Omron CX-Programmer project NewProject (CX-Programmer 9.66)

# PLC LQK19011ICM: CP1H XA
I/O table (CPU CP1H-XA40DR-A): rack 0 slot 0 CJ1W-SCU21

## Global symbols (name address type ; comment)
0.04 BOOL  ; SPARE
0.05 BOOL  ; SPARE
0.07 BOOL  ; VERTICAL.AXIS.DOWN.LIMT
0.08 BOOL  ; C0A
0.09 BOOL  ; C0B
0.11 BOOL  ; SAW.SOFT.START.FAULT
10 CHANNEL  ; Initialize the High Speed Encoder Channel to 0
100.00 BOOL  ; WATER.VALVE
100.01 BOOL  ; SOFT.START.RUN
100.02 BOOL  ; VERTICAL.AXIS.RAISE
100.03 BOOL  ; VERTICAL.AXIS.LOWER
100.04 BOOL  ; TRANSVERSE.AXIS.FORWARD
100.05 BOOL  ; TRANSVERSE.AXIS.REVERSE
100.06 BOOL  ; VERTICAL.AXIS.SPEED.SELECT
101.00 BOOL  ; SOFT.START.STOP
101.01 BOOL  ; ALARM
101.02 BOOL  ; LONG.AXIS.MASTER.DRV.INDEX.COMMAND
101.03 BOOL  ; VERTICAL.AXIS.BRAKE
101.04 BOOL  ; LONG.AXIS.MASTER.DRV.JOG.LEFT
101.05 BOOL  ; LONG.AXIS.MASTER.DRV.JOG.RIGHT
101.06 BOOL  ; LONG.AXIS.MASTER.DRV.INITIATE.HOME.MOVE
101.07 BOOL  ; LASER.ON
1.00 BOOL  ; WATER.FLOW.SWITCH
1.02 BOOL  ; SPARE
1.03 BOOL  ; PHOTOCELL_GAUCHE
1.04 BOOL  ; PHOTOCELL_DROIT
1.05 BOOL  ; TRANSVERSE.AXIS.HOME.PROXIMITY
1.06 BOOL  ; TRANSVERSE.AXIS.FORWARD.LIMT.PROXIMITY
1.07 BOOL  ; VERTICAL.AXIS.HOME.PROXIMITY
1.08 BOOL  ; VERTICAL.AXIS.FORWARD.LIMIT
1.12 BOOL  ; INCONNU
1.15 BOOL  ; DELETE
200 CHANNEL  ; ANALOG.INPUT1.SAW.CURRENT
210 CHANNEL  ; TRANSVERSE.AXIS.VELOCITY.REFERENCE
294 CHANNEL  ; RG3_FST_CUT
302 CHANNEL  ; Axis Long first Status Word
302.08 BOOL  ; LONG.AXIS.MASTER.STATUS.DRV.NEGLIM
302.09 BOOL  ; LONG.AXIS.MASTER.STATUS.DRV.POSLIM
302.13 BOOL  ; LONG.AXIS.MASTER.STATUS.DRV.JOGANYCMDCOMP
302.14 BOOL  ; LONG.AXIS.MASTER.STATUS.ABSPOSVAL
303 CHANNEL  ; Axis Long second status Word
303.00 BOOL  ; LONG.AXIS.MASTER.STATUS.DRV.INDEX0.LIMDISTHIT
303.01 BOOL  ; LONG.AXIS.MASTER.STATUS.DRV.INDEX0.CMD.INPRGRS
303.02 BOOL  ; LONG.AXIS.MASTER.STATUS.DRV.INDEX0.CMD.COMPLETE
303.03 BOOL  ; LONG.AXIS.MASTER.STATUS.DRV.INDEX0.PLSSTATUS
303.04 BOOL  ; LONG.AXIS.MASTER.STATUS.DRV.INDEX0.ACCELLERATING
303.05 BOOL  ; LONG.AXIS.MASTER.STATUS.DRV.INDEX0.ATVEL
303.06 BOOL  ; LONG.AXIS.MASTER.STATUS.DRV.INDEX0.DECELLERATING
303.07 BOOL  ; LONG.AXIS.MASTER.STATUS.DRV.INDEX.ANYCOMDCOMPLETE
303.08 BOOL  ; LONG.AXIS.MASTER.STATUS.DRV.PGMANYACTIVE
303.09 BOOL  ; LONG.AXIS.MASTER.STATUS.DRV.PGMANYCOMPLETE
303.10 BOOL  ; LONG.AXIS.MASTER.STATUS.DRV.PGM0.PGMRUNNING
303.11 BOOL  ; LONG.AXIS.MASTER.STATUS.DRV.PGM0.PGMCOMPLETE
304 CHANNEL  ; Axis Long third Status Word
304.00 BOOL  ; LONG.AXIS.MASTER.STATUS.DRV.ERROR.ERRORED
304.01 BOOL  ; LONG.AXIS.MASTER.STATUS.DRV.ERROR.SPDRIVETRIPACTIVE
304.02 BOOL  ; LONG.AXIS.MASTER.STATUS.DRV.ERROR.EZMOTION.WATCHDOG
304.03 BOOL  ; LONG.AXIS.MASTER.STATUS.DRV.ERROR.EZMOTION.INVALIDCONFIG
304.04 BOOL  ; LONG.AXIS.MASTER.STATUS.DRV.ERROR.EZMOTION.NVMINVALD
304.05 BOOL  ; LONG.AXIS.MASTER.STATUS.DRV.ERROR.EZMOTION.PWRUPTESTACTIVE
304.06 BOOL  ; LONG.AXIS.MASTER.STATUS.DRV.ERROR.EZMOTION.FOLLOWINGERRORACTIVE
304.07 BOOL  ; LONG.AXIS.MASTER.STATUS.DRV.ERROR.EZMOTION.TRAVLIMPLUSACTIVE
304.08 BOOL  ; LONG.AXIS.MASTER.STATUS.DRV.ERROR.EZMOTION.TRAVLIMNEGACTIVE
304.09 BOOL  ; LONG.AXIS.MASTER.STATUS.DRV.ERROR.EZMOTION.PGMERRORACTIVE
304.10 BOOL  ; LONG.AXIS.MASTER.STATUS.DRV.ERROR.EZMOTION.NOPRGACTIVE
304.11 BOOL  ; LONG.AXIS.MASTER.STATUS.DRV.EZMOTION.TRAJECTORYERRORACTIVE
304.12 BOOL  ; LONG.AXIS.MASTER.STATUS.DRV.EZMOTION.OUTPUTSHORTACTIVE
304.13 BOOL  ; LONG.AXIS.MASTER.STATUS.DRV.EZMOTION.CTNETERRORACTIVE
304.14 BOOL  ; LONG.AXIS.MASTER.STATUS.DRV.EZMOTION.OVERHEATACTIVE
304.15 BOOL  ; LONG.AXIS.MASTER.STATUS.DRV.EZMOTION.CAMERRORACTIVE
311 CHANNEL  ; Axis Long Control Word
311.00 BOOL  ; LONG.AXIS.MASTER.CONTROL.DRV.ERROR.RESET
311.03 BOOL  ; LONG.AXIS.MASTER.CONTROL.DRV.PGM0.INITIATE
311.04 BOOL  ; LONG.AXIS.MASTER.CONTROL.DRV.PGM0.STOP
311.05 BOOL  ; LONG.AXIS.MASTER.CONTROL.DRV.JOG.PLUS.ACTIVATE
311.06 BOOL  ; LONG.AXIS.MASTER.CONTROL.DRV.JOG.MINUS.ACTIVATE
600 CHANNEL  ; RG3_FST_CUT
D4 CHANNEL  ; Axis Command Distance
H0.02 BOOL  ; FIRST.CYCLE.COMPLETED
H10.02 BOOL  ; Axis Power Up Completed.
H10.03 BOOL  ; LONG.AXIS.DRIVE.ENO
H11.00 BOOL  ; VERTICAL.AXIS.POWER.OKAY
H11.01 BOOL  ; VERTICAL.AXIS.SAFETY.GATE.OKAY
H11.14 BOOL  ; VERTICAL.AXIS.ERROR.EXISTS
H11.15 BOOL  ; VERTICAL.AXIS.AUTO.OKAY
H12.00 BOOL  ; TRANSVERSE.AXIS.POWER.OKAY
H12.01 BOOL  ; TRANSVERSE.AXIS.SAFETY.GATE.OKAY
H12.14 BOOL  ; TRANSVERSE.AXIS.ERROR.EXISTS
H12.15 BOOL  ; TRANSVERSE.AXIS.AUTO.OKAY
W0.04 BOOL  ; SAFETY.GATE.OKAY
W10.01 BOOL  ; Axis Enable Complete
W10.05 BOOL  ; Axis Home Enabled
W10.06 BOOL  ; Axis Home Initiate Internal
W10.07 BOOL  ; Axis Home Active
W10.08 BOOL  ; Axis Home Complete
W10.09 BOOL  ; Axis Ref Enabled
W30.00 BOOL  ; OI.MESSAGE.INTERNAL.TRIGGER.MSG0
W30.01 BOOL  ; OI.MESSAGE.INTERNAL.TRIGGER.MSG1
W50.00 BOOL  ; SAFETY.GATE.CIRCUIT.OKAY
AxisPosition D5000 CHANNEL  ; Axis Actual Position Feedback from Drive
DRVERROR 0.01 BOOL  ; ANY.AXIS.ERROR
HSC0_Init HSC0_INIT
HSC0_PWR_INIT H0.00 BOOL  ; HSC 0 Power up Initialised
HSC1_Init HSC1_INIT
HSC1_PWR_INIT H0.01 BOOL  ; HSC 1 Power on Initialised
Home_Enable W0.15 BOOL  ; Homing Action Enable Global
IOTEMP W50 WORD  ; Word to hold temporary IO designations to be used in program in place of IO that have not been designated as yet.
LAXISMFDBK A276 CHANNEL  ; LONG.AXIS.MASTER,FEEDBACK
LAXISMFWDLIM 0.02 BOOL  ; LONG.AXIS.MASTER.FORWARD.LIMIT.PROXIMITY
MCR_ON 0.00 BOOL  ; MCR On, Control Power enabled
MC_Axis_Long_Drv_Disable 311.07 BOOL  ; LONG.AXIS.SOFT.DRIVE.DISABLE
MC_Axis_Long_Drv_Startup 302.01 BOOL  ; LONG.AXIS.MASTER.STATUS.DRV.STRTUP
MC_Axis_Long_En MC_Axis_En
MC_Axis_Long_Err H10.14 BOOL  ; LONG.AXIS.ERROR.EXISTS
MC_Axis_Long_Home MC_Axis_Home
MC_Axis_Long_Home_Cmd_Comp 302.15 BOOL  ; LONG.AXIS.MASTER.STATUS.DRV.HOME.ANYCMDCOMP
MC_Axis_Long_Home_Initiate 311.01 BOOL  ; LONG.AXIS.MASTER.CONTROL.DRV.HOME.INITIATE
MC_Axis_Long_Home_Sensor_Trig 311.02 BOOL  ; LONG.AXIS.MASTER.CONTROL.DRV.HOME0.SENSOR.TRIGGER
MC_Axis_Long_Pwr_Ok H10.00 BOOL  ; LONG.AXIS.POWER.OKAY
MC_Axis_Long_Ready_State H10.15 BOOL  ; Motion Control Status Ready State
MC_Axis_Long_Safety_Gate_Ok H10.01 BOOL  ; LONG.AXIS.SAFETY.GATE.OKAY
MC_Axis_Long_Status_Active 302.03 BOOL  ; LONG.AXIS.MASTER.STATUS.DRV.ACTIVE
MC_Axis_Long_Status_At_Vel 302.06 BOOL  ; LONG.AXIS.MASTER.STATUS.DRV.ATVEL
MC_Axis_Long_Status_En 302.00 BOOL  ; LONG.AXIS.MASTER.STATUS.DRV.EN
MC_Axis_Long_Status_Healthy 302.04 BOOL  ; LONG.AXIS.MASTER.STATUS.DRV.HEALTHY
MC_Axis_Long_Status_In_Pos 302.07 BOOL  ; LONG.AXIS.MASTER.STATUS.DRV.INPOS
MC_Axis_Long_Status_Ok 302.02 BOOL  ; LONG.AXIS.MASTER.STATUS.DRV.OK
MC_Axis_Status_Cmd_Motion 302.05 BOOL  ; LONG.AXIS.MASTER.STATUS.DRV.STARTUP
MC_Internal_Axis_Long_En_Req W10.00 BOOL  ; AxisRefComplete
MC_Internal_Axis_Long_Err W10.14 BOOL  ; MC_Internal_Axis_Long_Err
OICTRLAUTOMSTOP W120.03 BOOL  ; OI.CONTROL.AUTOMATIC.CYCLE.MACHINE.STOP
OICTRLAUTOSTART W120.02 BOOL  ; OI.CONTROL.AUTOMATIC.CYCLE.START
OICTRLAUTOSTOP W120.01 BOOL  ; OI.CONTROL.AUTOMATIC.CYCLE.STOP
OICTRLHASEL W120.00 BOOL  ; OI.CONTROL.HAND.AUTO.SELECTOR
OIMSGCLR W101 INT  ; OI.MESSAGE.COLOUR
OIMSGSEL W100 INT  ; OI.MESSAGE.SELECT
Power_On W0.03 BOOL  ; Main Power is on and first cycle is completed
Transverse_Axis_Feedback A272 CHANNEL  ; Transverse axis positonal feedback from incremental encoder mounted on motor
Transverse_Axis_Home_Completed H0.11 BOOL  ; Transverse Axis Homing Completed
Transverse_Home_Request W1.02 BOOL  ; Transverse axis home request
Transverse_Homing H1.01 BOOL  ; Transverse Axis Homing
Vertical_Axis_Feedback A270 CHANNEL  ; Vertical axis position feedback from incremental encoder mounted on motor
Vertical_Home_Complete H0.10 BOOL  ; Vertical Axis Homing Completed
Vertical_Homing H1.00 BOOL  ; Vertical Axis Homing
Vertical_Homing_Request W0.02 BOOL  ; Vertical axis home action request.

## Program Main (cyclic task 0)
; Main saw program file
Local symbols
Channel_for_HSC0 INT  ; The Default Channel for HSC 0
HSC0_Init_Plx W0.00 BOOL  ; HSC0 Initialised at Power Up
HSC1_Init_Plx W1.00 BOOL  ; HSC1 Initialised at power up
Long_Axis_En_Request BOOL

### Section Init_HSC

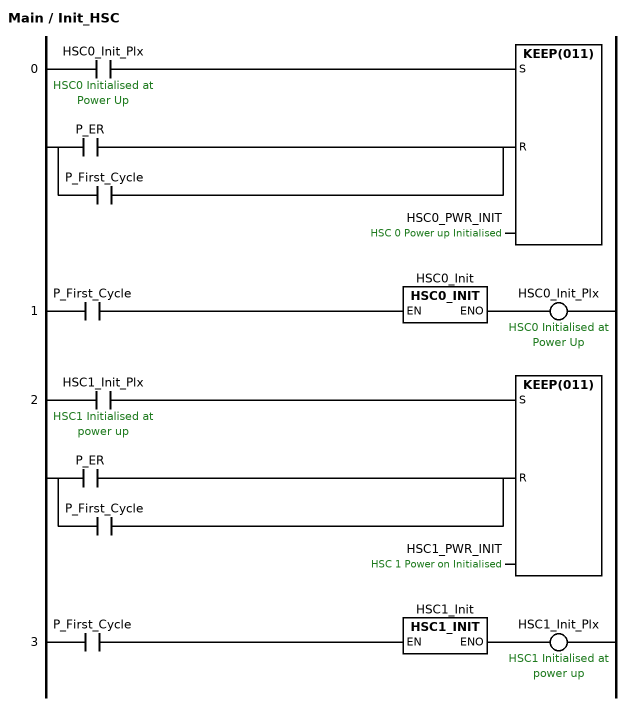
; rung 0
LD HSC0_Init_Plx  ; HSC0 Initialised at Power Up
LD P_ER
OR P_First_Cycle
KEEP(011) HSC0_PWR_INIT  ; HSC 0 Power up Initialised
; rung 1
LD P_First_Cycle
CALL HSC0_Init : HSC0_INIT ()
OUT HSC0_Init_Plx  ; HSC0 Initialised at Power Up
; rung 2
LD HSC1_Init_Plx  ; HSC1 Initialised at power up
LD P_ER
OR P_First_Cycle
KEEP(011) HSC1_PWR_INIT  ; HSC 1 Power on Initialised
; rung 3
LD P_First_Cycle
CALL HSC1_Init : HSC1_INIT ()
OUT HSC1_Init_Plx  ; HSC1 Initialised at power up

### Section Init_Power

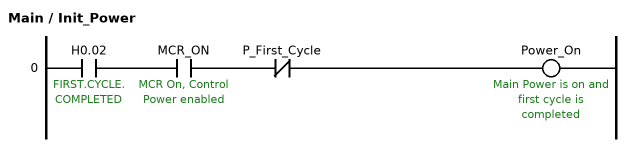
; rung 0
LD H0.02  ; FIRST.CYCLE.COMPLETED
AND MCR_ON  ; MCR On, Control Power enabled
ANDNOT P_First_Cycle
OUT Power_On  ; Main Power is on and first cycle is completed

### Section Init_Safety

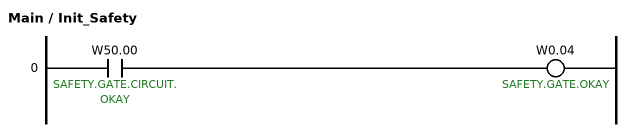
; rung 0
LD W50.00  ; SAFETY.GATE.CIRCUIT.OKAY
OUT W0.04  ; SAFETY.GATE.OKAY

### Section Init_Long_Axis

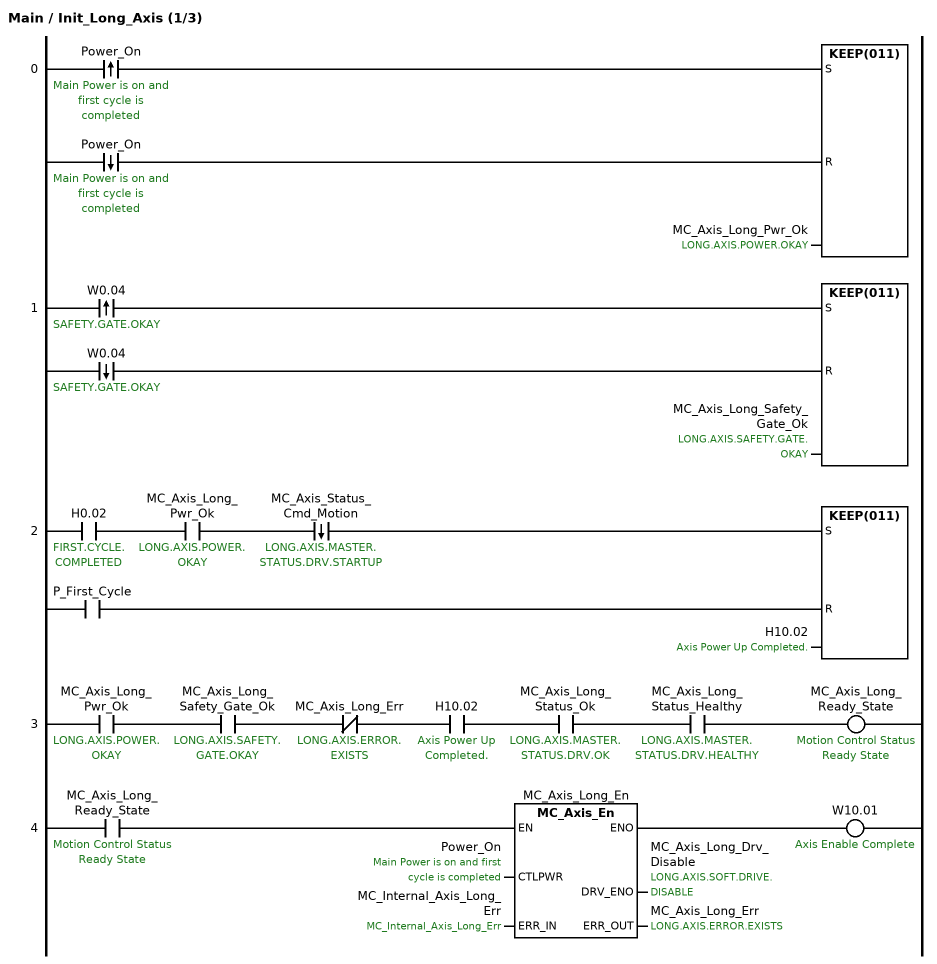
; rung 0
@LD Power_On  ; Main Power is on and first cycle is completed
%LD Power_On  ; Main Power is on and first cycle is completed
KEEP(011) MC_Axis_Long_Pwr_Ok  ; LONG.AXIS.POWER.OKAY
; rung 1
@LD W0.04  ; SAFETY.GATE.OKAY
%LD W0.04  ; SAFETY.GATE.OKAY
KEEP(011) MC_Axis_Long_Safety_Gate_Ok  ; LONG.AXIS.SAFETY.GATE.OKAY
; rung 2
LD H0.02  ; FIRST.CYCLE.COMPLETED
AND MC_Axis_Long_Pwr_Ok  ; LONG.AXIS.POWER.OKAY
%AND MC_Axis_Status_Cmd_Motion  ; LONG.AXIS.MASTER.STATUS.DRV.STARTUP
LD P_First_Cycle
KEEP(011) H10.02  ; Axis Power Up Completed.
; rung 3
LD MC_Axis_Long_Pwr_Ok  ; LONG.AXIS.POWER.OKAY
AND MC_Axis_Long_Safety_Gate_Ok  ; LONG.AXIS.SAFETY.GATE.OKAY
ANDNOT MC_Axis_Long_Err  ; LONG.AXIS.ERROR.EXISTS
AND H10.02  ; Axis Power Up Completed.
AND MC_Axis_Long_Status_Ok  ; LONG.AXIS.MASTER.STATUS.DRV.OK
AND MC_Axis_Long_Status_Healthy  ; LONG.AXIS.MASTER.STATUS.DRV.HEALTHY
OUT MC_Axis_Long_Ready_State  ; Motion Control Status Ready State
; rung 4
LD MC_Axis_Long_Ready_State  ; Motion Control Status Ready State
CALL MC_Axis_Long_En : MC_Axis_En (CTLPWR := Power_On, ERR_IN := MC_Internal_Axis_Long_Err, DRV_ENO => MC_Axis_Long_Drv_Disable, ERR_OUT => MC_Axis_Long_Err)  ; Main Power is on and first cycle is completed, MC_Internal_Axis_Long_Err, LONG.AXIS.SOFT.DRIVE.DISABLE, LONG.AXIS.ERROR.EXISTS
OUT W10.01  ; Axis Enable Complete

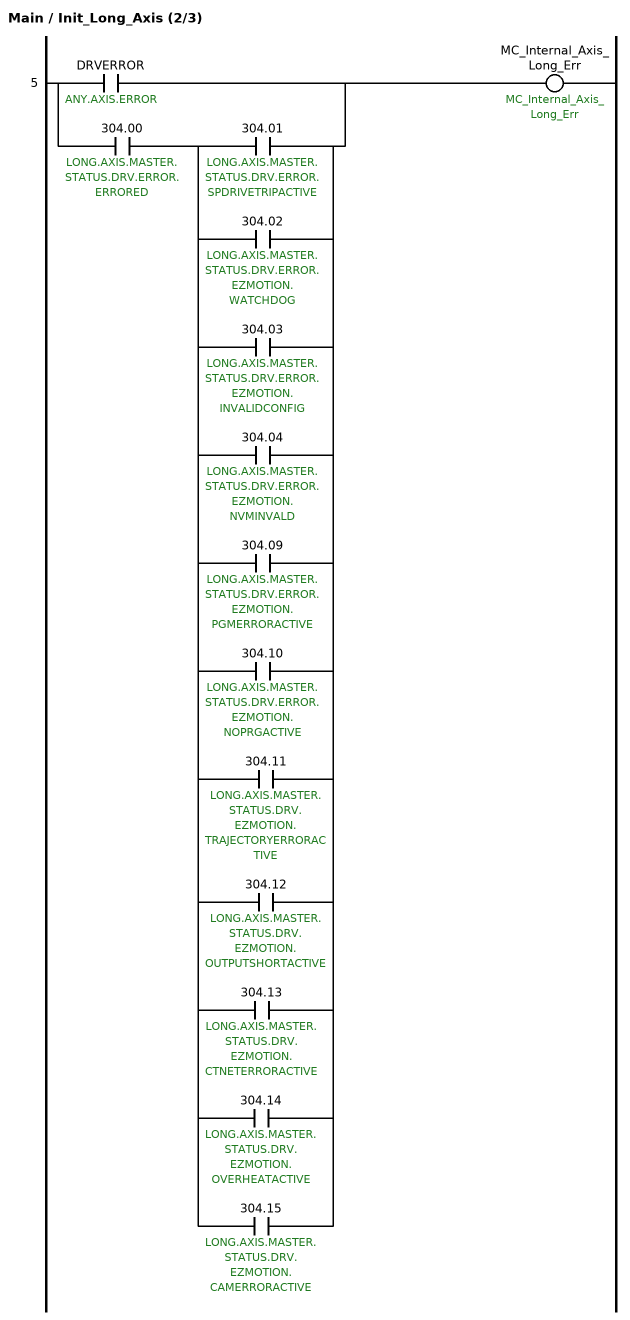
; rung 5
LD DRVERROR  ; ANY.AXIS.ERROR
LD 304.00  ; LONG.AXIS.MASTER.STATUS.DRV.ERROR.ERRORED
LD 304.01  ; LONG.AXIS.MASTER.STATUS.DRV.ERROR.SPDRIVETRIPACTIVE
OR 304.02  ; LONG.AXIS.MASTER.STATUS.DRV.ERROR.EZMOTION.WATCHDOG
OR 304.03  ; LONG.AXIS.MASTER.STATUS.DRV.ERROR.EZMOTION.INVALIDCONFIG
OR 304.04  ; LONG.AXIS.MASTER.STATUS.DRV.ERROR.EZMOTION.NVMINVALD
OR 304.09  ; LONG.AXIS.MASTER.STATUS.DRV.ERROR.EZMOTION.PGMERRORACTIVE
OR 304.10  ; LONG.AXIS.MASTER.STATUS.DRV.ERROR.EZMOTION.NOPRGACTIVE
OR 304.11  ; LONG.AXIS.MASTER.STATUS.DRV.EZMOTION.TRAJECTORYERRORACTIVE
OR 304.12  ; LONG.AXIS.MASTER.STATUS.DRV.EZMOTION.OUTPUTSHORTACTIVE
OR 304.13  ; LONG.AXIS.MASTER.STATUS.DRV.EZMOTION.CTNETERRORACTIVE
OR 304.14  ; LONG.AXIS.MASTER.STATUS.DRV.EZMOTION.OVERHEATACTIVE
OR 304.15  ; LONG.AXIS.MASTER.STATUS.DRV.EZMOTION.CAMERRORACTIVE
ANDLD
ORLD
OUT MC_Internal_Axis_Long_Err  ; MC_Internal_Axis_Long_Err

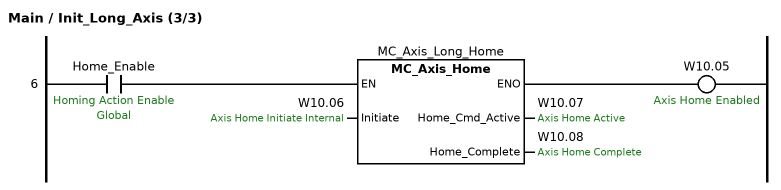
; rung 6
LD Home_Enable  ; Homing Action Enable Global
CALL MC_Axis_Long_Home : MC_Axis_Home (Initiate := W10.06, Home_Cmd_Active => W10.07, Home_Complete => W10.08)  ; Axis Home Initiate Internal, Axis Home Active, Axis Home Complete
OUT W10.05  ; Axis Home Enabled

### Section Init_Vertical_Axis

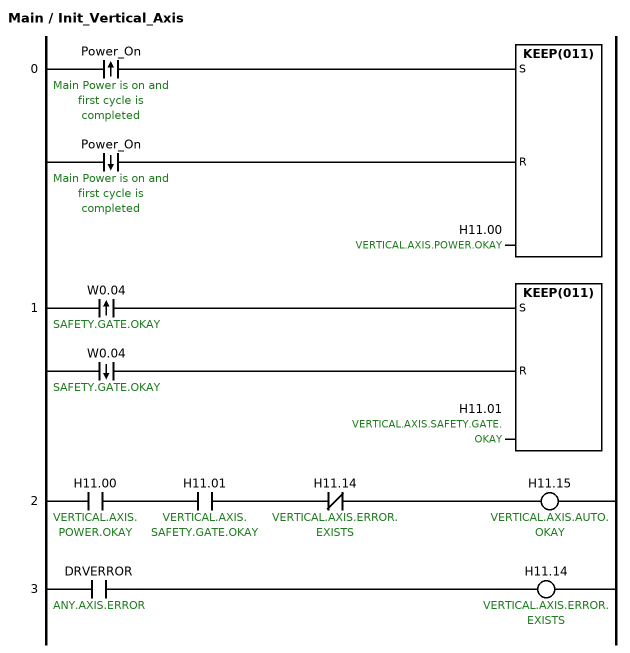
; rung 0
@LD Power_On  ; Main Power is on and first cycle is completed
%LD Power_On  ; Main Power is on and first cycle is completed
KEEP(011) H11.00  ; VERTICAL.AXIS.POWER.OKAY
; rung 1
@LD W0.04  ; SAFETY.GATE.OKAY
%LD W0.04  ; SAFETY.GATE.OKAY
KEEP(011) H11.01  ; VERTICAL.AXIS.SAFETY.GATE.OKAY
; rung 2
LD H11.00  ; VERTICAL.AXIS.POWER.OKAY
AND H11.01  ; VERTICAL.AXIS.SAFETY.GATE.OKAY
ANDNOT H11.14  ; VERTICAL.AXIS.ERROR.EXISTS
OUT H11.15  ; VERTICAL.AXIS.AUTO.OKAY
; rung 3
LD DRVERROR  ; ANY.AXIS.ERROR
OUT H11.14  ; VERTICAL.AXIS.ERROR.EXISTS

### Section Init_Transverse_Axis

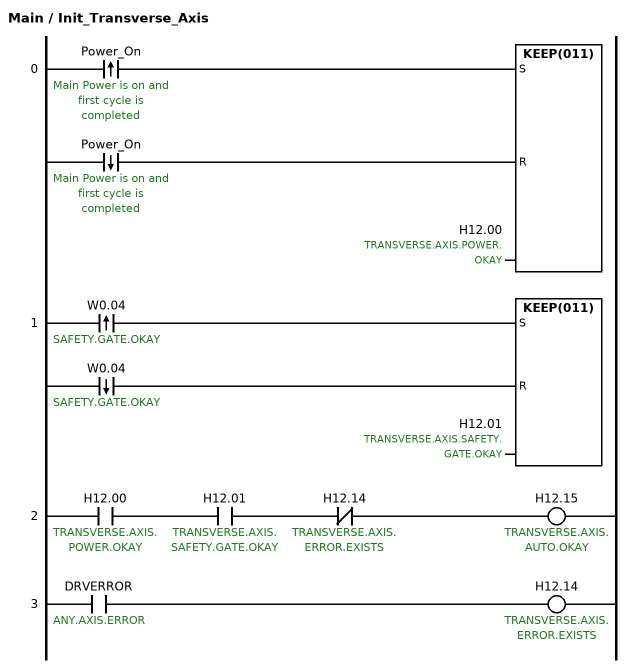
; rung 0
@LD Power_On  ; Main Power is on and first cycle is completed
%LD Power_On  ; Main Power is on and first cycle is completed
KEEP(011) H12.00  ; TRANSVERSE.AXIS.POWER.OKAY
; rung 1
@LD W0.04  ; SAFETY.GATE.OKAY
%LD W0.04  ; SAFETY.GATE.OKAY
KEEP(011) H12.01  ; TRANSVERSE.AXIS.SAFETY.GATE.OKAY
; rung 2
LD H12.00  ; TRANSVERSE.AXIS.POWER.OKAY
AND H12.01  ; TRANSVERSE.AXIS.SAFETY.GATE.OKAY
ANDNOT H12.14  ; TRANSVERSE.AXIS.ERROR.EXISTS
OUT H12.15  ; TRANSVERSE.AXIS.AUTO.OKAY
; rung 3
LD DRVERROR  ; ANY.AXIS.ERROR
OUT H12.14  ; TRANSVERSE.AXIS.ERROR.EXISTS

### Section Init_Message_Display

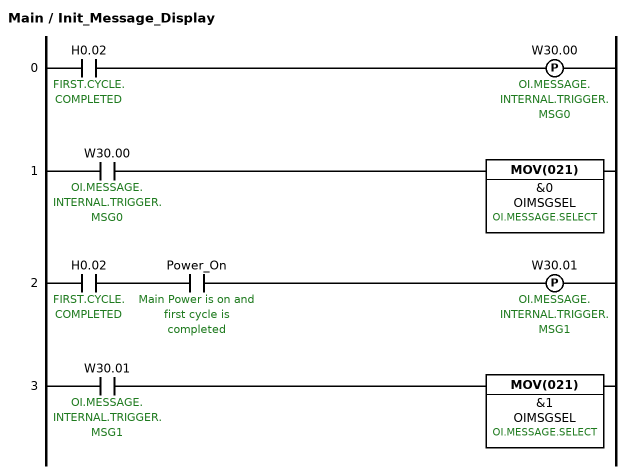
; rung 0
LD H0.02  ; FIRST.CYCLE.COMPLETED
DIFU(013) W30.00  ; OI.MESSAGE.INTERNAL.TRIGGER.MSG0
; rung 1
LD W30.00  ; OI.MESSAGE.INTERNAL.TRIGGER.MSG0
MOV(021) &0 OIMSGSEL  ; OI.MESSAGE.SELECT
; rung 2
LD H0.02  ; FIRST.CYCLE.COMPLETED
AND Power_On  ; Main Power is on and first cycle is completed
DIFU(013) W30.01  ; OI.MESSAGE.INTERNAL.TRIGGER.MSG1
; rung 3
LD W30.01  ; OI.MESSAGE.INTERNAL.TRIGGER.MSG1
MOV(021) &1 OIMSGSEL  ; OI.MESSAGE.SELECT

### Section END

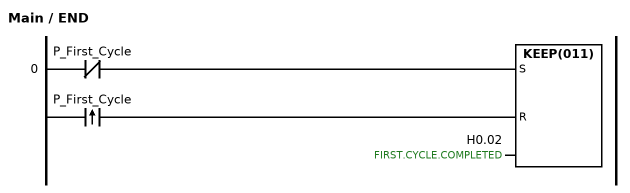
; rung 0
LDNOT P_First_Cycle
@LD P_First_Cycle
KEEP(011) H0.02  ; FIRST.CYCLE.COMPLETED
; rung 1
END(001)

## Function block HSC0_INIT
; Initialise HSC Channel Selected
VAR
  Preset : DINT;
END_VAR

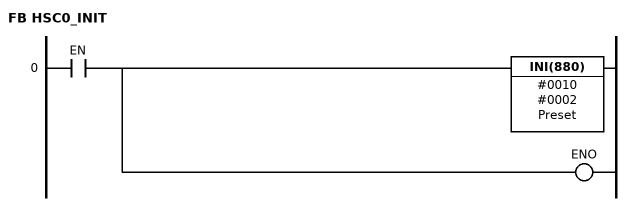
; rung 0
LD EN
INI(880) #0010 #0002 Preset
OUT ENO

## Function block HSC1_INIT
; Initialise HSC Channel Selected
VAR
  Preset : DINT;
END_VAR

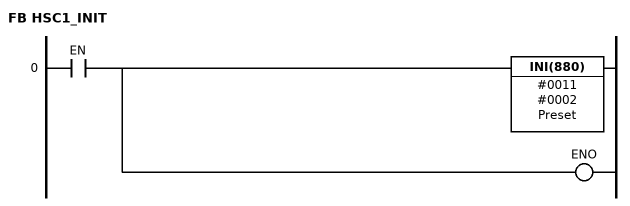
; rung 0
LD EN
INI(880) #0011 #0002 Preset
OUT ENO

## Function block MC_Axis_En
; Function Block for enabling Drives used in motion control.
VAR_INPUT
  CTLPWR : BOOL;
  ERR_IN : BOOL;
END_VAR
VAR_OUTPUT
  DRV_ENO : BOOL;  (* Drive Enable Output. *)
  ERR_OUT : BOOL;  (* Drive Error Output. *)
END_VAR
VAR_EXTERNAL
  Power_On AT W0.03 : BOOL;
  MC_Internal_Axis_Long_Err AT W10.14 : BOOL;
END_VAR
(*This Function Block is intended for use with VFD's in a motion application.*)
ENO :=  EN; (*Turn on the Enable Output if Block is enabled*)
IF CTLPWR = TRUE  THEN
	DRV_ENO :=  FALSE;(*DRV_ENO is connected to the drive disable soft command and needs inversion*)
	IF ERR_IN = FALSE THEN
		ERR_OUT :=  FALSE;
	ELSE ERR_OUT := TRUE;
		DRV_ENO := TRUE;
	END_IF;
ELSE DRV_ENO := TRUE;
END_IF;

## Function block MC_Axis_Home
VAR_INPUT
  Initiate : BOOL;  (* Initiate Homing Sequence *)
END_VAR
VAR_OUTPUT
  Home_Cmd_Active : BOOL;  (* Homing Command is Active *)
  Home_Complete : BOOL;  (* Homing Command Complete *)
END_VAR
VAR_EXTERNAL
  MC_Axis_Long_Home_Initiate AT 311.01 : BOOL;  (* LONG.AXIS.MASTER.CONTROL.DRV.HOME.INITIATE *)
  MC_Axis_Long_Home_Sensor_Trig AT 311.02 : BOOL;  (* LONG.AXIS.MASTER.CONTROL.DRV.HOME0.SENSOR.TRIGGER *)
  MC_Axis_Long_Home_Cmd_Comp AT 302.15 : BOOL;  (* LONG.AXIS.MASTER.STATUS.DRV.HOME.ANYCMDCOMP *)
  MC_Axis_Status_Cmd_Motion AT 302.05 : BOOL;  (* LONG.AXIS.MASTER.STATUS.DRV.CMDMOTION *)
  MC_Axis_Long_Status_In_Pos AT 302.07 : BOOL;  (* LONG.AXIS.MASTER.STATUS.DRV.INPOS *)
END_VAR
(*Function Block to be used for motion control Homing function*)
ENO:= EN;
IF Initiate = TRUE THEN
	MC_Axis_Long_Home_Initiate:= TRUE;
	IF MC_Axis_Status_Cmd_Motion=TRUE THEN
		Home_Cmd_Active:= TRUE;
	END_IF;
ELSE
	MC_Axis_Long_Home_Initiate:= FALSE;
END_IF;
IF MC_Axis_Long_Home_Cmd_Comp = TRUE THEN
	Home_Cmd_Active:= FALSE;
	Home_Complete:= TRUE;
ELSE Home_Complete:= FALSE;
END_IF;